{attribute addProperty BoxType "EL9110-0000-0016"}
{attribute addProperty Id "PowerOKAT %I*PowerOK_E4AEF59E810WcStateAT %I*WcState_98A4DF7520.250InfoDataAT %I*InfoData_192954DE1620"}
{attribute addProperty CRC "913442673"}
{attribute addProperty SizeInBites "26"}
{attribute addProperty SizeInBytes "3.25"}
TYPE EL9110_AE5731BA :
STRUCT
	{attribute addProperty Name "PowerOK"}
	PowerOK : PowerOK_E4AEF59E;
	{attribute addProperty Name "WcState"}
	WcState : WcState_98A4DF75;
	{attribute addProperty Name "InfoData"}
	InfoData : InfoData_192954DE;
END_STRUCT
END_TYPE

(* stored: Version 1.2.0.0, ProductVersion 3.1.4024.9
   DUT EL9110_AE5731BA: Id {64360e27-2059-471a-a617-0e05c095877f} *)
